    |   movel([0.574480, -1.254823, -2.655022, -0.802544, 1.570796, 2.145277],accel_mss,speed_ms,0,blend_radius_m)
    |   movel([0.572653, -1.256207, -2.654278, -0.801904, 1.570796, 2.143449],accel_mss,speed_ms,0,blend_radius_m)
    |   movel([0.570903, -1.257701, -2.653472, -0.801216, 1.570796, 2.141699],accel_mss,speed_ms,0,blend_radius_m)
    |   speed_ms = 0.005
    |   movel([0.570903, -1.248125, -2.648928, -0.815336, 1.570796, 2.141699],accel_mss,speed_ms,0,blend_radius_m)
    |   speed_ms = 0.040
    |   movel([0.581833, -1.236261, -2.655167, -0.820961, 1.570796, 2.152630],accel_mss,speed_ms,0,blend_radius_m)
    |   speed_ms = 0.005
    |   movel([0.581833, -1.245895, -2.659765, -0.806729, 1.570796, 2.152630],accel_mss,speed_ms,0,blend_radius_m)
    |   speed_ms = 0.025
    |   movel([0.580655, -1.245118, -2.660174, -0.807098, 1.570796, 2.151451],accel_mss,speed_ms,0,blend_radius_m)
    |   movel([0.579245, -1.244644, -2.660422, -0.807323, 1.570796, 2.150042],accel_mss,speed_ms,0,blend_radius_m)
    |   movel([0.577646, -1.244456, -2.660521, -0.807412, 1.570796, 2.148442],accel_mss,speed_ms,0,blend_radius_m)
    |   movel([0.575895, -1.244521, -2.660487, -0.807381, 1.570796, 2.146691],accel_mss,speed_ms,0,blend_radius_m)
    |   movel([0.574029, -1.244817, -2.660332, -0.807240, 1.570796, 2.144826],accel_mss,speed_ms,0,blend_radius_m)
    |   movel([0.572093, -1.245317, -2.660069, -0.807003, 1.570796, 2.142889],accel_mss,speed_ms,0,blend_radius_m)
    |   movel([0.570122, -1.245989, -2.659716, -0.806684, 1.570796, 2.140919],accel_mss,speed_ms,0,blend_radius_m)
    |   movel([0.568160, -1.246811, -2.659283, -0.806295, 1.570796, 2.138956],accel_mss,speed_ms,0,blend_radius_m)
    |   movel([0.566149, -1.247795, -2.658764, -0.805830, 1.570796, 2.136945],accel_mss,speed_ms,0,blend_radius_m)
    |   movel([0.564149, -1.248921, -2.658168, -0.805300, 1.570796, 2.134946],accel_mss,speed_ms,0,blend_radius_m)
    |   movel([0.562186, -1.250182, -2.657499, -0.804707, 1.570796, 2.132982],accel_mss,speed_ms,0,blend_radius_m)
    |   movel([0.560295, -1.251575, -2.656759, -0.804056, 1.570796, 2.131091],accel_mss,speed_ms,0,blend_radius_m)
    |   movel([0.558508, -1.253085, -2.655953, -0.803352, 1.570796, 2.129305],accel_mss,speed_ms,0,blend_radius_m)
    |   movel([0.556856, -1.254705, -2.655085, -0.802599, 1.570796, 2.127652],accel_mss,speed_ms,0,blend_radius_m)
    |   movel([0.555373, -1.256431, -2.654157, -0.801801, 1.570796, 2.126169],accel_mss,speed_ms,0,blend_radius_m)
    |   movel([0.554087, -1.258250, -2.653175, -0.800964, 1.570796, 2.124883],accel_mss,speed_ms,0,blend_radius_m)
    |   speed_ms = 0.005
    |   movel([0.554087, -1.248676, -2.648634, -0.815079, 1.570796, 2.124883],accel_mss,speed_ms,0,blend_radius_m)
    |   speed_ms = 0.040
    |   movel([0.560669, -1.236787, -2.654894, -0.820708, 1.570796, 2.131465],accel_mss,speed_ms,0,blend_radius_m)
    |   speed_ms = 0.005
    |   movel([0.560669, -1.246418, -2.659490, -0.806481, 1.570796, 2.131465],accel_mss,speed_ms,0,blend_radius_m)
    |   speed_ms = 0.025
    |   movel([0.558095, -1.246749, -2.659315, -0.806324, 1.570796, 2.128891],accel_mss,speed_ms,0,blend_radius_m)
    |   movel([0.555260, -1.247449, -2.658946, -0.805994, 1.570796, 2.126057],accel_mss,speed_ms,0,blend_radius_m)
    |   movel([0.552301, -1.248510, -2.658386, -0.805493, 1.570796, 2.123097],accel_mss,speed_ms,0,blend_radius_m)
    |   movel([0.549355, -1.249923, -2.657637, -0.804829, 1.570796, 2.120151],accel_mss,speed_ms,0,blend_radius_m)
    |   movel([0.546557, -1.251678, -2.656704, -0.804007, 1.570796, 2.117353],accel_mss,speed_ms,0,blend_radius_m)
    |   movel([0.545253, -1.252682, -2.656168, -0.803539, 1.570796, 2.116050],accel_mss,speed_ms,0,blend_radius_m)
    |   movel([0.544040, -1.253765, -2.655589, -0.803035, 1.570796, 2.114836],accel_mss,speed_ms,0,blend_radius_m)
    |   movel([0.542928, -1.254931, -2.654964, -0.802494, 1.570796, 2.113724],accel_mss,speed_ms,0,blend_radius_m)
    |   movel([0.541935, -1.256174, -2.654296, -0.801920, 1.570796, 2.112732],accel_mss,speed_ms,0,blend_radius_m)
    |   movel([0.541083, -1.257492, -2.653585, -0.801312, 1.570796, 2.111880],accel_mss,speed_ms,0,blend_radius_m)
    |   movel([0.540381, -1.258889, -2.652830, -0.800671, 1.570796, 2.111177],accel_mss,speed_ms,0,blend_radius_m)
    |   speed_ms = 0.005
    |   movel([0.540381, -1.249318, -2.648291, -0.814780, 1.570796, 2.111177],accel_mss,speed_ms,0,blend_radius_m)
    |   speed_ms = 0.040
    |   movel([0.539729, -1.243401, -2.651432, -0.817556, 1.570796, 2.110525],accel_mss,speed_ms,0,blend_radius_m)
    |   speed_ms = 0.005
    |   movel([0.539729, -1.253001, -2.655998, -0.803391, 1.570796, 2.110525],accel_mss,speed_ms,0,blend_radius_m)
    |   speed_ms = 0.025
    |   movel([0.535561, -1.255244, -2.654796, -0.802350, 1.570796, 2.106357],accel_mss,speed_ms,0,blend_radius_m)
    |   movel([0.533496, -1.256537, -2.654100, -0.801752, 1.570796, 2.104292],accel_mss,speed_ms,0,blend_radius_m)
    |   movel([0.531501, -1.257950, -2.653338, -0.801101, 1.570796, 2.102298],accel_mss,speed_ms,0,blend_radius_m)
    |   movel([0.529616, -1.259495, -2.652501, -0.800393, 1.570796, 2.100412],accel_mss,speed_ms,0,blend_radius_m)
    |   movel([0.527876, -1.261180, -2.651586, -0.799624, 1.570796, 2.098673],accel_mss,speed_ms,0,blend_radius_m)
    |   movel([0.526329, -1.263009, -2.650587, -0.798792, 1.570796, 2.097126],accel_mss,speed_ms,0,blend_radius_m)
    |   movel([0.525007, -1.264994, -2.649500, -0.797895, 1.570796, 2.095803],accel_mss,speed_ms,0,blend_radius_m)
    |   speed_ms = 0.005
    |   # Splitting Linear movement in 2 (instruction 3386: MoveL 3110)
    |   movel([0.525007, -1.241553, -2.638115, -0.832721, 1.570796, 2.095803],accel_mss,speed_ms,0,blend_radius_m)
    |   movel([0.525007, -1.219449, -2.626381, -0.866560, 1.570796, 2.095803],accel_mss,speed_ms,0,blend_radius_m)
    |   speed_ms = 1.000
    |   movel([0.525007, -1.219449, -2.626381, -0.866560, 1.570796, 2.095803],accel_mss,speed_ms,0,blend_radius_m)
    |   # Splitting Linear movement in 6 (instruction 3389: MoveL 3112)
    |   movel([0.525007, -1.185458, -2.606099, -0.920831, 1.570796, 2.095803],accel_mss,speed_ms,0,blend_radius_m)
    |   movel([0.525007, -1.154843, -2.584985, -0.972561, 1.570796, 2.095803],accel_mss,speed_ms,0,blend_radius_m)
    |   movel([0.525007, -1.127379, -2.563110, -1.021900, 1.570796, 2.095803],accel_mss,speed_ms,0,blend_radius_m)
    |   movel([0.525007, -1.102846, -2.540541, -1.069003, 1.570796, 2.095803],accel_mss,speed_ms,0,blend_radius_m)
    |   movel([0.525007, -1.081028, -2.517332, -1.114030, 1.570796, 2.095803],accel_mss,speed_ms,0,blend_radius_m)
    |   movel([0.525007, -1.061721, -2.493532, -1.157137, 1.570796, 2.095803],accel_mss,speed_ms,0,blend_radius_m)
    |   # End of main program
    | end
    | 
    | Machining4()
